PROGRAM PRG_LARS_ValidationAsConfirmation
VAR
	rtrigNewOuterArrived					: R_TRIG;
	bNewOuterIsProccesing				: BOOL;
	tonValidationTimout					: TON;
	bValidationTimeout					: BOOL;
	bValidationTimeoutReset				: BOOL;
	fbTimeoutCounter						: CTU;
	nCount									: WORD;
	fbPerformance							: FB_Interval;

	bOuterValidationCameraTrigger			: BOOL;
	aOuterValidationCamera				:  ARRAY[1..2] OF FB_SCANNER_CameraSelect;
	stOuterValidationCameraStatus		: ST_SCANNER;
	(*stOuterValidationCameraOptions		: ST_SCANNER_Options := (eScannerType := E_MV_420_FULL, nImageBuffer := 1, nExpectedResp := 2);*)
	aOuterValidationEvaluation			: ARRAY[1..2] OF FB_SCANNER_Evaluation;

	fbValidationCameraOut				: FB_OUTER_ValidationCameraOut;
	fbCheckForDuplicateOuterValidation	: FB_OUTER_CheckDuplicateStatus;

	(*rtrigOuterValidationCameraDone		: R_TRIG;
	bOuterValidationCameraDone			: BOOL;*)
	bDataReadyForValidation				: BOOL;
	bQAReject								: BOOL;

	sLastImageLableString				: T_OUTER_Barcode;

	fbMoveOuterData						: FB_OUTER_MoveOuterStatus;
	fbCompleteDataFromConfirmation	: FB_OUTER_CompleteDataFromDB_SingleCam;
	fbMETSValidateOuterForReject			: FB_OUTER_ValidateOuterForReject;
	tofValidateOuterDoneForHMI			: TOF;
	fbMasterListUpdate					: FB_OUTER_MasterListUpdate;

	stLastOuterCompleted					: ST_OUTER_Status;
	sLastReadOuterBarcode				: T_OUTER_Barcode;
	sLastReadConfPackCode1				: T_PACK_Barcode;
	nOutersCompleted						: UDINT;
	bDoneInfo								: BOOL;

	rtrigSetOuterValidationOK			: R_TRIG;
	rtrigSetOuterValidationNOK		: R_TRIG;

	rsOuterRejectStation 				: RS;
	rsOuterRejectConfirmation 		: RS;

	rtrigResetValidationStatus			: R_TRIG;

	sRejectCode						: STRING(255);
	fbArchiveInvalidOuters			: FB_OUTER_ArchiveInvalidOuters;
	aReasonForReject					: ARRAY[0..50] OF STRING(255);
	bClearList							: BOOL;

	fbOuterProduced					: FB_KPI_GenericEfficiency;
	fbOuterInspection					: FB_KPI_OutersEfficiency;

	fbOuterLevelCounter				: FB_KPI_OuterLevelCounter;

	fbQARejectCounter				: FB_CTU32;
	fbOuterValidationIndexOK			: FB_CTU32;

	ctuConsecutiveOuterRejects		: CTU;
	nActualCount						: WORD;

	stDummyImageData			: ST_SCANNER_ImageData;		(* image data structure *)
	aDistanceCheck				: ARRAY[1..2] OF FB_TimeDistance;
	bResetCTU						: BOOL;
END_VAR
VAR // added by the converter: edge detectors and wires of the graphical bodies
    _w1 : BOOL;
END_VAR

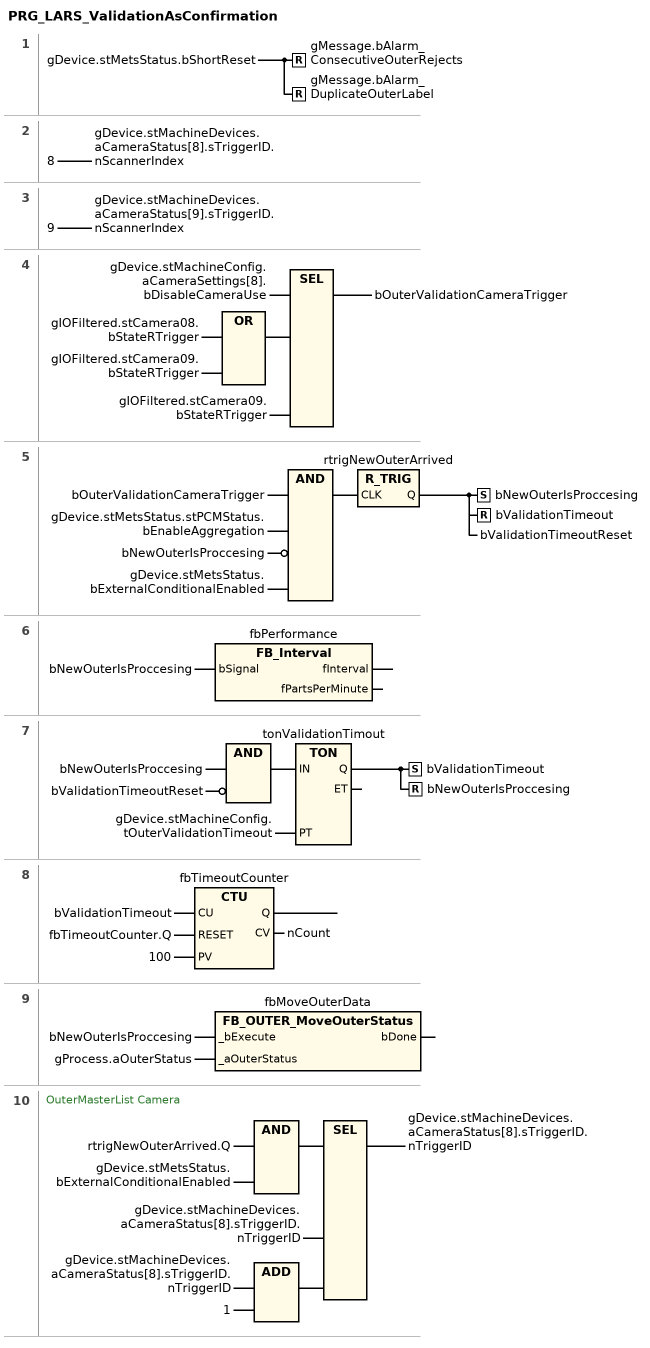
// NETWORK 1
gMessage.bAlarm_ConsecutiveOuterRejects R= gDevice.stMetsStatus.bShortReset;
gMessage.bAlarm_DuplicateOuterLabel R= gDevice.stMetsStatus.bShortReset;

// NETWORK 2
gDevice.stMachineDevices.aCameraStatus[8].sTriggerID.nScannerIndex := 8;

// NETWORK 3
gDevice.stMachineDevices.aCameraStatus[9].sTriggerID.nScannerIndex := 9;

// NETWORK 4
bOuterValidationCameraTrigger := SEL(gDevice.stMachineConfig.aCameraSettings[8].bDisableCameraUse, gIOFiltered.stCamera08.bStateRTrigger OR gIOFiltered.stCamera09.bStateRTrigger, gIOFiltered.stCamera09.bStateRTrigger);

// NETWORK 5
rtrigNewOuterArrived(CLK := bOuterValidationCameraTrigger AND gDevice.stMetsStatus.stPCMStatus.bEnableAggregation AND NOT bNewOuterIsProccesing AND gDevice.stMetsStatus.bExternalConditionalEnabled); // R_TRIG
bNewOuterIsProccesing S= rtrigNewOuterArrived.Q;
bValidationTimeout R= rtrigNewOuterArrived.Q;
bValidationTimeoutReset := rtrigNewOuterArrived.Q;

// NETWORK 6
fbPerformance(bSignal := bNewOuterIsProccesing); // FB_Interval

// NETWORK 7
tonValidationTimout(IN := bNewOuterIsProccesing AND NOT bValidationTimeoutReset, PT := gDevice.stMachineConfig.tOuterValidationTimeout); // TON
bValidationTimeout S= tonValidationTimout.Q;
bNewOuterIsProccesing R= tonValidationTimout.Q;

// NETWORK 8
fbTimeoutCounter(CU := bValidationTimeout, RESET := fbTimeoutCounter.Q, PV := 100, CV => nCount); // CTU

// NETWORK 9
fbMoveOuterData(_bExecute := bNewOuterIsProccesing, _aOuterStatus := gProcess.aOuterStatus); // FB_OUTER_MoveOuterStatus

// NETWORK 10
// OuterMasterList Camera
gDevice.stMachineDevices.aCameraStatus[8].sTriggerID.nTriggerID := SEL(rtrigNewOuterArrived.Q AND gDevice.stMetsStatus.bExternalConditionalEnabled, gDevice.stMachineDevices.aCameraStatus[8].sTriggerID.nTriggerID, gDevice.stMachineDevices.aCameraStatus[8].sTriggerID.nTriggerID + 1);

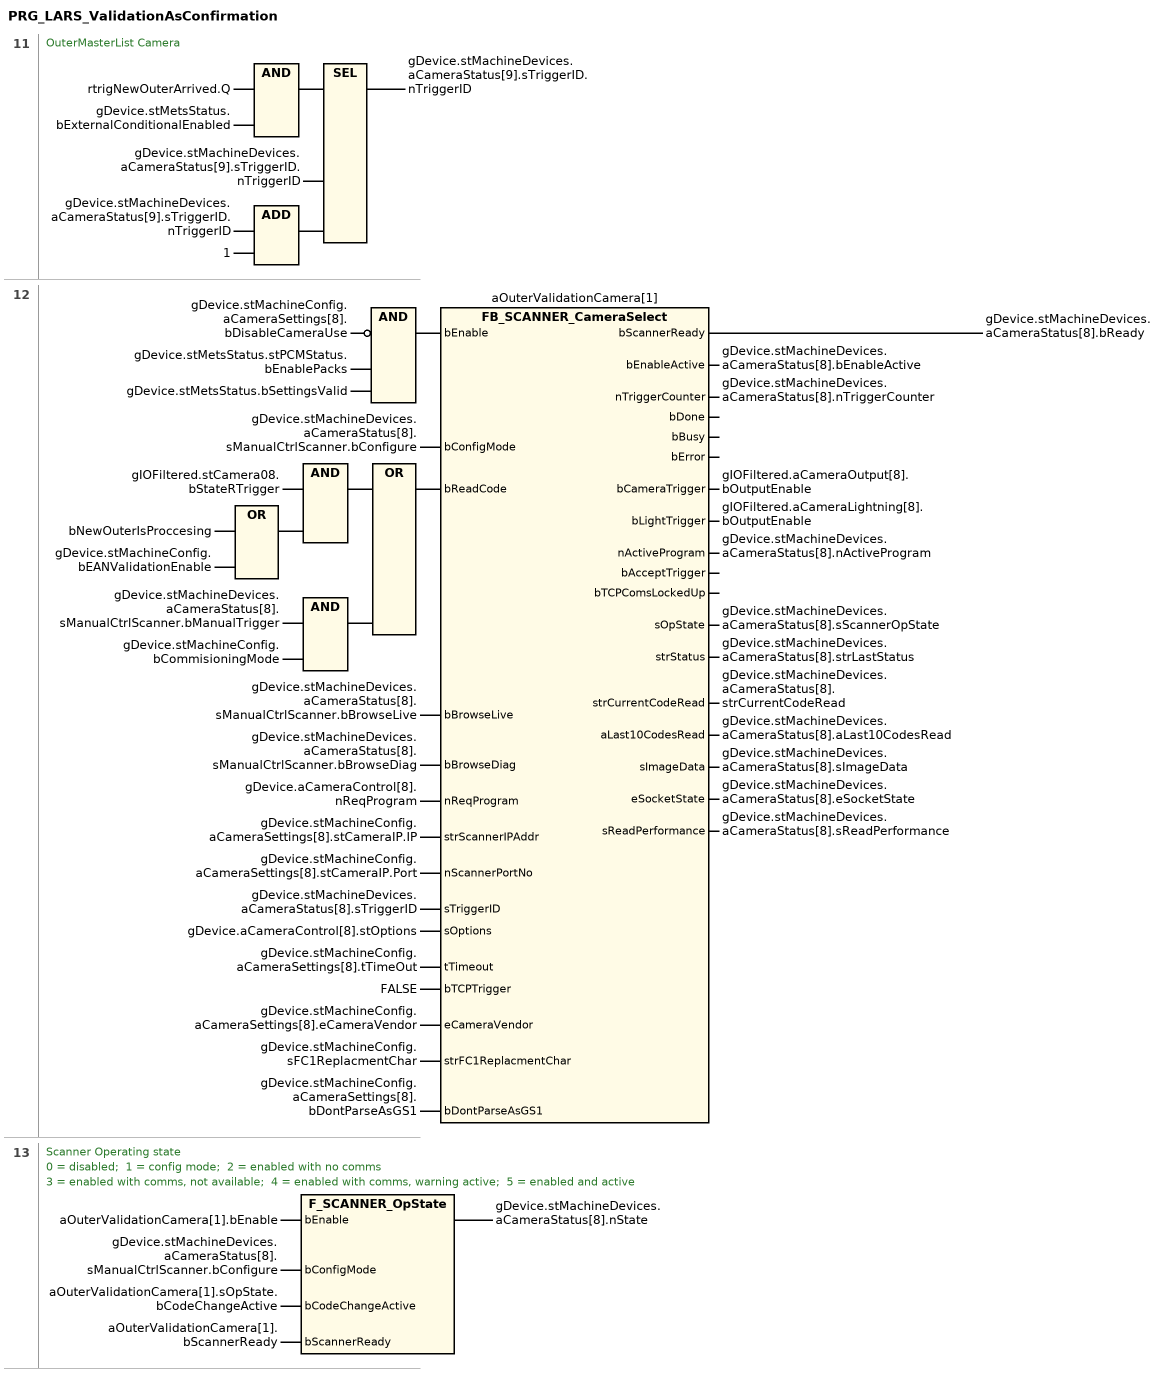
// NETWORK 11
// OuterMasterList Camera
gDevice.stMachineDevices.aCameraStatus[9].sTriggerID.nTriggerID := SEL(rtrigNewOuterArrived.Q AND gDevice.stMetsStatus.bExternalConditionalEnabled, gDevice.stMachineDevices.aCameraStatus[9].sTriggerID.nTriggerID, gDevice.stMachineDevices.aCameraStatus[9].sTriggerID.nTriggerID + 1);

// NETWORK 12
aOuterValidationCamera[1](
    bEnable := NOT gDevice.stMachineConfig.aCameraSettings[8].bDisableCameraUse AND gDevice.stMetsStatus.stPCMStatus.bEnablePacks AND gDevice.stMetsStatus.bSettingsValid,
    bConfigMode := gDevice.stMachineDevices.aCameraStatus[8].sManualCtrlScanner.bConfigure,
    bReadCode := gIOFiltered.stCamera08.bStateRTrigger AND (bNewOuterIsProccesing OR gDevice.stMachineConfig.bEANValidationEnable) OR gDevice.stMachineDevices.aCameraStatus[8].sManualCtrlScanner.bManualTrigger AND gDevice.stMachineConfig.bCommisioningMode,
    bBrowseLive := gDevice.stMachineDevices.aCameraStatus[8].sManualCtrlScanner.bBrowseLive,
    bBrowseDiag := gDevice.stMachineDevices.aCameraStatus[8].sManualCtrlScanner.bBrowseDiag,
    nReqProgram := gDevice.aCameraControl[8].nReqProgram,
    strScannerIPAddr := gDevice.stMachineConfig.aCameraSettings[8].stCameraIP.IP,
    nScannerPortNo := gDevice.stMachineConfig.aCameraSettings[8].stCameraIP.Port,
    sTriggerID := gDevice.stMachineDevices.aCameraStatus[8].sTriggerID,
    sOptions := gDevice.aCameraControl[8].stOptions,
    tTimeout := gDevice.stMachineConfig.aCameraSettings[8].tTimeOut,
    bTCPTrigger := FALSE,
    eCameraVendor := gDevice.stMachineConfig.aCameraSettings[8].eCameraVendor,
    strFC1ReplacmentChar := gDevice.stMachineConfig.sFC1ReplacmentChar,
    bDontParseAsGS1 := gDevice.stMachineConfig.aCameraSettings[8].bDontParseAsGS1,
    bEnableActive => gDevice.stMachineDevices.aCameraStatus[8].bEnableActive,
    nTriggerCounter => gDevice.stMachineDevices.aCameraStatus[8].nTriggerCounter,
    bCameraTrigger => gIOFiltered.aCameraOutput[8].bOutputEnable,
    bLightTrigger => gIOFiltered.aCameraLightning[8].bOutputEnable,
    nActiveProgram => gDevice.stMachineDevices.aCameraStatus[8].nActiveProgram,
    sOpState => gDevice.stMachineDevices.aCameraStatus[8].sScannerOpState,
    strStatus => gDevice.stMachineDevices.aCameraStatus[8].strLastStatus,
    strCurrentCodeRead => gDevice.stMachineDevices.aCameraStatus[8].strCurrentCodeRead,
    aLast10CodesRead => gDevice.stMachineDevices.aCameraStatus[8].aLast10CodesRead,
    sImageData => gDevice.stMachineDevices.aCameraStatus[8].sImageData,
    eSocketState => gDevice.stMachineDevices.aCameraStatus[8].eSocketState,
    sReadPerformance => gDevice.stMachineDevices.aCameraStatus[8].sReadPerformance); // FB_SCANNER_CameraSelect
gDevice.stMachineDevices.aCameraStatus[8].bReady := aOuterValidationCamera[1].bScannerReady;

// NETWORK 13
// 					Scanner Operating state
// 0 = disabled;  1 = config mode;  2 = enabled with no comms
// 3 = enabled with comms, not available;  4 = enabled with comms, warning active;  5 = enabled and active
//
gDevice.stMachineDevices.aCameraStatus[8].nState := F_SCANNER_OpState(bEnable := aOuterValidationCamera[1].bEnable, bConfigMode := gDevice.stMachineDevices.aCameraStatus[8].sManualCtrlScanner.bConfigure, bCodeChangeActive := aOuterValidationCamera[1].sOpState.bCodeChangeActive, bScannerReady := aOuterValidationCamera[1].bScannerReady);

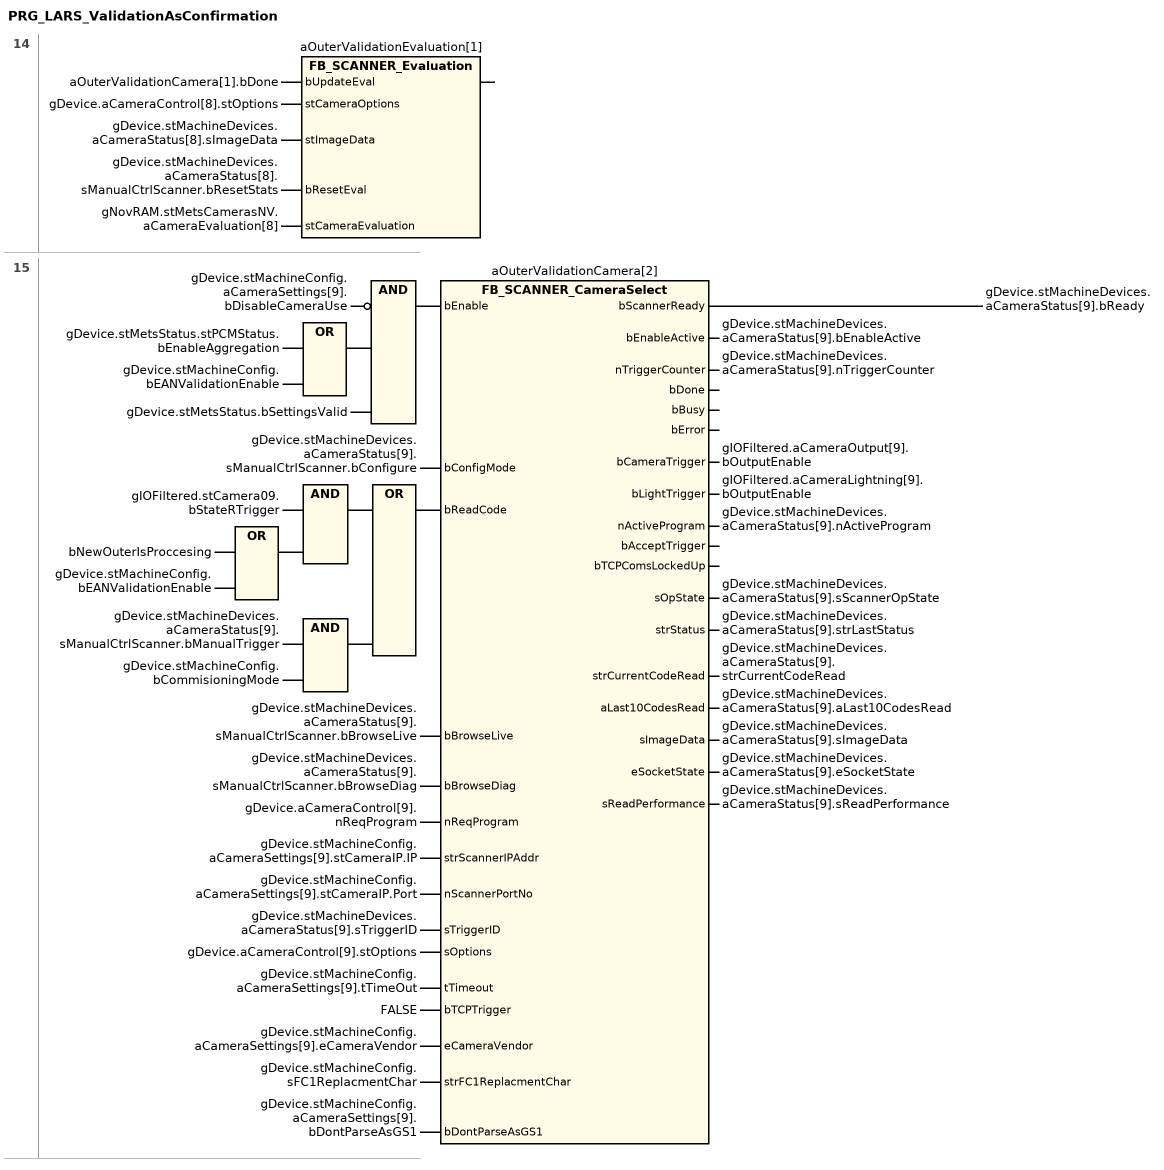
// NETWORK 14
aOuterValidationEvaluation[1](
    bUpdateEval := aOuterValidationCamera[1].bDone,
    stCameraOptions := gDevice.aCameraControl[8].stOptions,
    stImageData := gDevice.stMachineDevices.aCameraStatus[8].sImageData,
    bResetEval := gDevice.stMachineDevices.aCameraStatus[8].sManualCtrlScanner.bResetStats,
    stCameraEvaluation := gNovRAM.stMetsCamerasNV.aCameraEvaluation[8]); // FB_SCANNER_Evaluation

// NETWORK 15
aOuterValidationCamera[2](
    bEnable := NOT gDevice.stMachineConfig.aCameraSettings[9].bDisableCameraUse AND (gDevice.stMetsStatus.stPCMStatus.bEnableAggregation OR gDevice.stMachineConfig.bEANValidationEnable) AND gDevice.stMetsStatus.bSettingsValid,
    bConfigMode := gDevice.stMachineDevices.aCameraStatus[9].sManualCtrlScanner.bConfigure,
    bReadCode := gIOFiltered.stCamera09.bStateRTrigger AND (bNewOuterIsProccesing OR gDevice.stMachineConfig.bEANValidationEnable) OR gDevice.stMachineDevices.aCameraStatus[9].sManualCtrlScanner.bManualTrigger AND gDevice.stMachineConfig.bCommisioningMode,
    bBrowseLive := gDevice.stMachineDevices.aCameraStatus[9].sManualCtrlScanner.bBrowseLive,
    bBrowseDiag := gDevice.stMachineDevices.aCameraStatus[9].sManualCtrlScanner.bBrowseDiag,
    nReqProgram := gDevice.aCameraControl[9].nReqProgram,
    strScannerIPAddr := gDevice.stMachineConfig.aCameraSettings[9].stCameraIP.IP,
    nScannerPortNo := gDevice.stMachineConfig.aCameraSettings[9].stCameraIP.Port,
    sTriggerID := gDevice.stMachineDevices.aCameraStatus[9].sTriggerID,
    sOptions := gDevice.aCameraControl[9].stOptions,
    tTimeout := gDevice.stMachineConfig.aCameraSettings[9].tTimeOut,
    bTCPTrigger := FALSE,
    eCameraVendor := gDevice.stMachineConfig.aCameraSettings[9].eCameraVendor,
    strFC1ReplacmentChar := gDevice.stMachineConfig.sFC1ReplacmentChar,
    bDontParseAsGS1 := gDevice.stMachineConfig.aCameraSettings[9].bDontParseAsGS1,
    bEnableActive => gDevice.stMachineDevices.aCameraStatus[9].bEnableActive,
    nTriggerCounter => gDevice.stMachineDevices.aCameraStatus[9].nTriggerCounter,
    bCameraTrigger => gIOFiltered.aCameraOutput[9].bOutputEnable,
    bLightTrigger => gIOFiltered.aCameraLightning[9].bOutputEnable,
    nActiveProgram => gDevice.stMachineDevices.aCameraStatus[9].nActiveProgram,
    sOpState => gDevice.stMachineDevices.aCameraStatus[9].sScannerOpState,
    strStatus => gDevice.stMachineDevices.aCameraStatus[9].strLastStatus,
    strCurrentCodeRead => gDevice.stMachineDevices.aCameraStatus[9].strCurrentCodeRead,
    aLast10CodesRead => gDevice.stMachineDevices.aCameraStatus[9].aLast10CodesRead,
    sImageData => gDevice.stMachineDevices.aCameraStatus[9].sImageData,
    eSocketState => gDevice.stMachineDevices.aCameraStatus[9].eSocketState,
    sReadPerformance => gDevice.stMachineDevices.aCameraStatus[9].sReadPerformance); // FB_SCANNER_CameraSelect
gDevice.stMachineDevices.aCameraStatus[9].bReady := aOuterValidationCamera[2].bScannerReady;

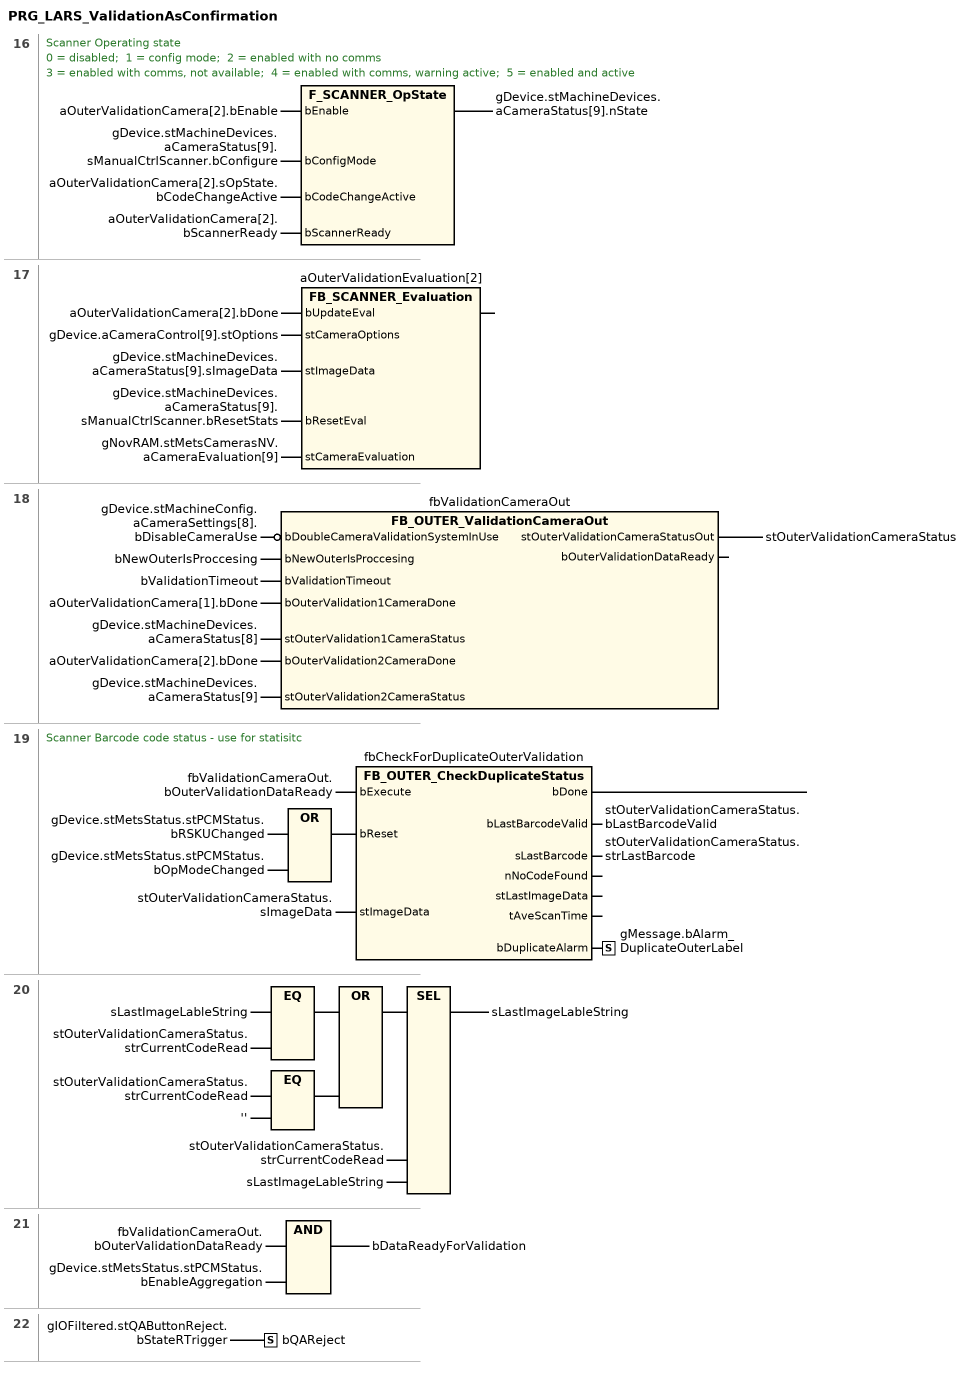
// NETWORK 16
// 					Scanner Operating state
// 0 = disabled;  1 = config mode;  2 = enabled with no comms
// 3 = enabled with comms, not available;  4 = enabled with comms, warning active;  5 = enabled and active
//
gDevice.stMachineDevices.aCameraStatus[9].nState := F_SCANNER_OpState(bEnable := aOuterValidationCamera[2].bEnable, bConfigMode := gDevice.stMachineDevices.aCameraStatus[9].sManualCtrlScanner.bConfigure, bCodeChangeActive := aOuterValidationCamera[2].sOpState.bCodeChangeActive, bScannerReady := aOuterValidationCamera[2].bScannerReady);

// NETWORK 17
aOuterValidationEvaluation[2](
    bUpdateEval := aOuterValidationCamera[2].bDone,
    stCameraOptions := gDevice.aCameraControl[9].stOptions,
    stImageData := gDevice.stMachineDevices.aCameraStatus[9].sImageData,
    bResetEval := gDevice.stMachineDevices.aCameraStatus[9].sManualCtrlScanner.bResetStats,
    stCameraEvaluation := gNovRAM.stMetsCamerasNV.aCameraEvaluation[9]); // FB_SCANNER_Evaluation

// NETWORK 18
fbValidationCameraOut(
    bDoubleCameraValidationSystemInUse := NOT gDevice.stMachineConfig.aCameraSettings[8].bDisableCameraUse,
    bNewOuterIsProccesing := bNewOuterIsProccesing,
    bValidationTimeout := bValidationTimeout,
    bOuterValidation1CameraDone := aOuterValidationCamera[1].bDone,
    stOuterValidation1CameraStatus := gDevice.stMachineDevices.aCameraStatus[8],
    bOuterValidation2CameraDone := aOuterValidationCamera[2].bDone,
    stOuterValidation2CameraStatus := gDevice.stMachineDevices.aCameraStatus[9]); // FB_OUTER_ValidationCameraOut
stOuterValidationCameraStatus := fbValidationCameraOut.stOuterValidationCameraStatusOut;

// NETWORK 19
// Scanner Barcode code status - use for statisitc
fbCheckForDuplicateOuterValidation(
    bExecute := fbValidationCameraOut.bOuterValidationDataReady,
    bReset := gDevice.stMetsStatus.stPCMStatus.bRSKUChanged OR gDevice.stMetsStatus.stPCMStatus.bOpModeChanged,
    stImageData := stOuterValidationCameraStatus.sImageData,
    bLastBarcodeValid => stOuterValidationCameraStatus.bLastBarcodeValid,
    sLastBarcode => stOuterValidationCameraStatus.strLastBarcode); // FB_OUTER_CheckDuplicateStatus
gMessage.bAlarm_DuplicateOuterLabel S= fbCheckForDuplicateOuterValidation.bDuplicateAlarm;

// NETWORK 20
sLastImageLableString := SEL(sLastImageLableString = stOuterValidationCameraStatus.strCurrentCodeRead OR stOuterValidationCameraStatus.strCurrentCodeRead = '', stOuterValidationCameraStatus.strCurrentCodeRead, sLastImageLableString);

// NETWORK 21
bDataReadyForValidation := fbValidationCameraOut.bOuterValidationDataReady AND gDevice.stMetsStatus.stPCMStatus.bEnableAggregation;

// NETWORK 22
bQAReject S= gIOFiltered.stQAButtonReject.bStateRTrigger;

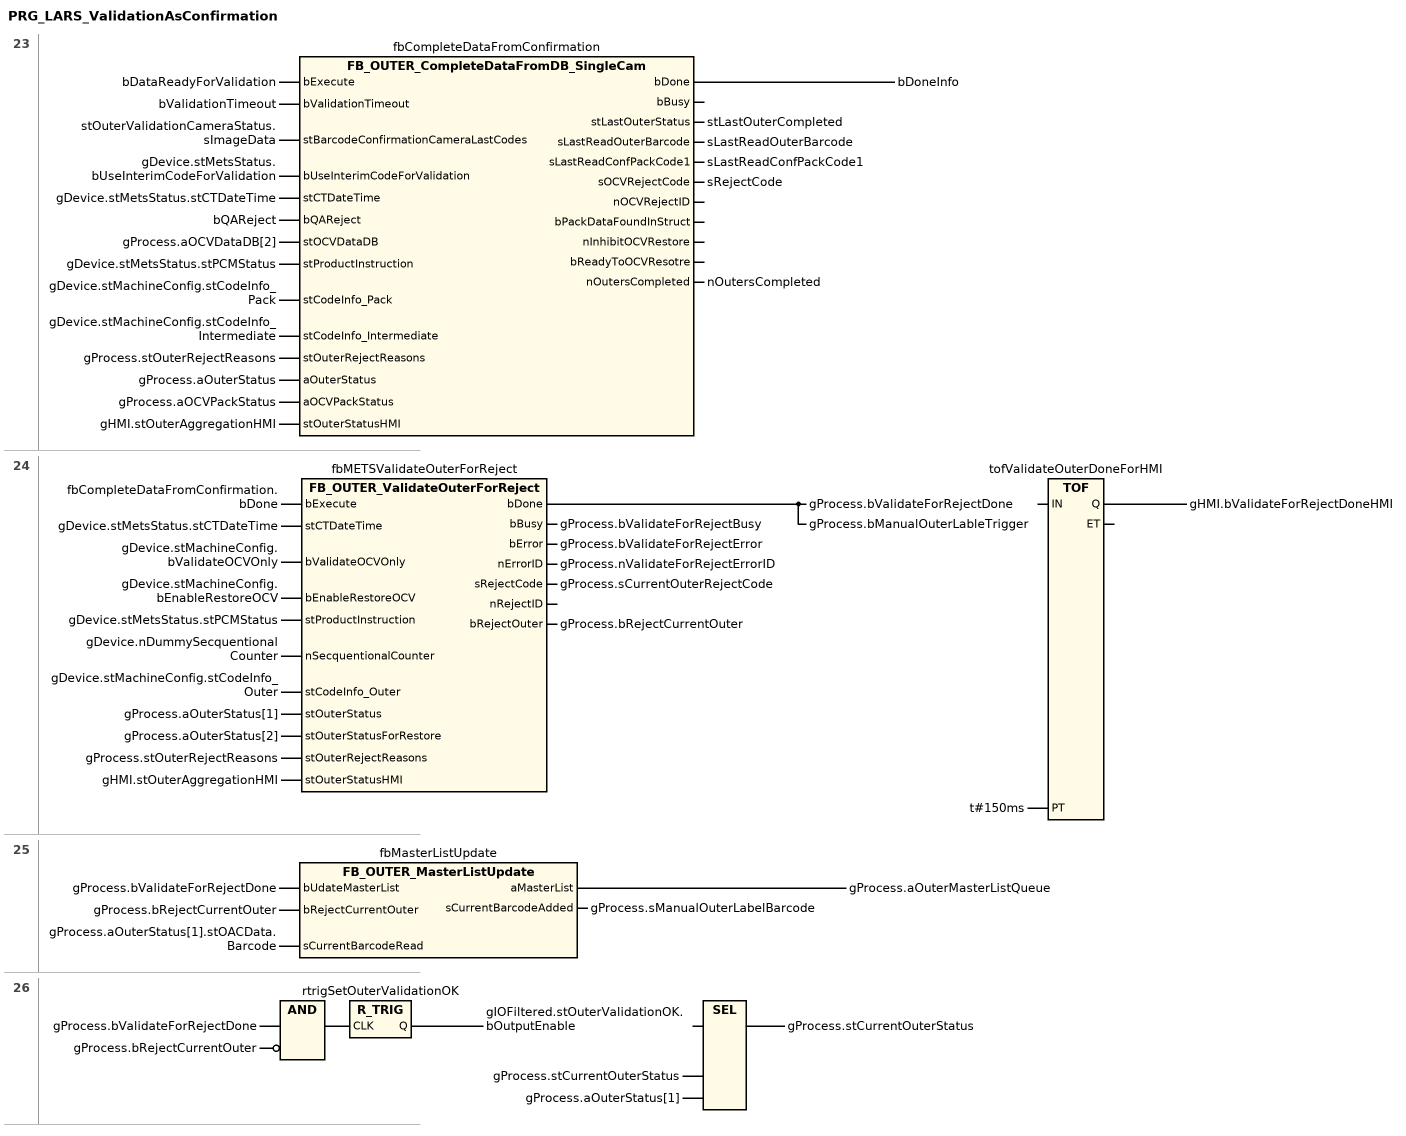
// NETWORK 23
fbCompleteDataFromConfirmation(
    bExecute := bDataReadyForValidation,
    bValidationTimeout := bValidationTimeout,
    stBarcodeConfirmationCameraLastCodes := stOuterValidationCameraStatus.sImageData,
    bUseInterimCodeForValidation := gDevice.stMetsStatus.bUseInterimCodeForValidation,
    stCTDateTime := gDevice.stMetsStatus.stCTDateTime,
    bQAReject := bQAReject,
    stOCVDataDB := gProcess.aOCVDataDB[2],
    stProductInstruction := gDevice.stMetsStatus.stPCMStatus,
    stCodeInfo_Pack := gDevice.stMachineConfig.stCodeInfo_Pack,
    stCodeInfo_Intermediate := gDevice.stMachineConfig.stCodeInfo_Intermediate,
    stOuterRejectReasons := gProcess.stOuterRejectReasons,
    aOuterStatus := gProcess.aOuterStatus,
    aOCVPackStatus := gProcess.aOCVPackStatus,
    stOuterStatusHMI := gHMI.stOuterAggregationHMI,
    stLastOuterStatus => stLastOuterCompleted,
    sLastReadOuterBarcode => sLastReadOuterBarcode,
    sLastReadConfPackCode1 => sLastReadConfPackCode1,
    sOCVRejectCode => sRejectCode,
    nOutersCompleted => nOutersCompleted); // FB_OUTER_CompleteDataFromDB_SingleCam
bDoneInfo := fbCompleteDataFromConfirmation.bDone;

// NETWORK 24
fbMETSValidateOuterForReject(
    bExecute := fbCompleteDataFromConfirmation.bDone,
    stCTDateTime := gDevice.stMetsStatus.stCTDateTime,
    bValidateOCVOnly := gDevice.stMachineConfig.bValidateOCVOnly,
    bEnableRestoreOCV := gDevice.stMachineConfig.bEnableRestoreOCV,
    stProductInstruction := gDevice.stMetsStatus.stPCMStatus,
    nSecquentionalCounter := gDevice.nDummySecquentionalCounter,
    stCodeInfo_Outer := gDevice.stMachineConfig.stCodeInfo_Outer,
    stOuterStatus := gProcess.aOuterStatus[1],
    stOuterStatusForRestore := gProcess.aOuterStatus[2],
    stOuterRejectReasons := gProcess.stOuterRejectReasons,
    stOuterStatusHMI := gHMI.stOuterAggregationHMI,
    bBusy => gProcess.bValidateForRejectBusy,
    bError => gProcess.bValidateForRejectError,
    nErrorID => gProcess.nValidateForRejectErrorID,
    sRejectCode => gProcess.sCurrentOuterRejectCode,
    bRejectOuter => gProcess.bRejectCurrentOuter); // FB_OUTER_ValidateOuterForReject
gProcess.bValidateForRejectDone := fbMETSValidateOuterForReject.bDone;
gProcess.bManualOuterLableTrigger := fbMETSValidateOuterForReject.bDone;
tofValidateOuterDoneForHMI(IN := fbMETSValidateOuterForReject.bDone, PT := t#150ms); // TOF
gHMI.bValidateForRejectDoneHMI := tofValidateOuterDoneForHMI.Q;

// NETWORK 25
fbMasterListUpdate(
    bUdateMasterList := gProcess.bValidateForRejectDone,
    bRejectCurrentOuter := gProcess.bRejectCurrentOuter,
    sCurrentBarcodeRead := gProcess.aOuterStatus[1].stOACData.Barcode,
    sCurrentBarcodeAdded => gProcess.sManualOuterLabelBarcode); // FB_OUTER_MasterListUpdate
gProcess.aOuterMasterListQueue := fbMasterListUpdate.aMasterList;

// NETWORK 26
rtrigSetOuterValidationOK(CLK := gProcess.bValidateForRejectDone AND NOT gProcess.bRejectCurrentOuter); // R_TRIG
gIOFiltered.stOuterValidationOK.bOutputEnable := rtrigSetOuterValidationOK.Q;
gProcess.stCurrentOuterStatus := SEL(rtrigSetOuterValidationOK.Q, gProcess.stCurrentOuterStatus, gProcess.aOuterStatus[1]);

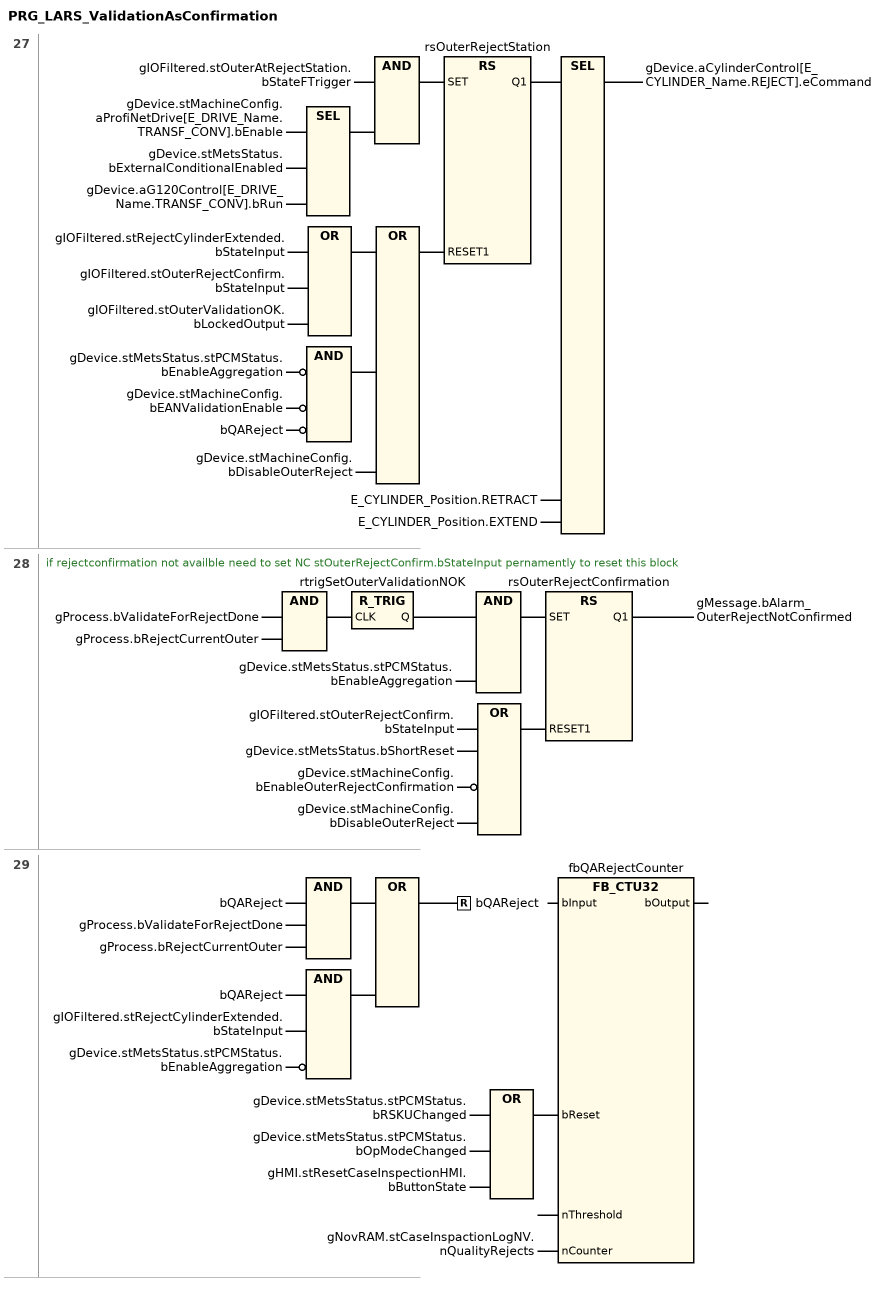
// NETWORK 27
rsOuterRejectStation(SET := gIOFiltered.stOuterAtRejectStation.bStateFTrigger AND SEL(gDevice.stMachineConfig.aProfiNetDrive[E_DRIVE_Name.TRANSF_CONV].bEnable, gDevice.stMetsStatus.bExternalConditionalEnabled, gDevice.aG120Control[E_DRIVE_Name.TRANSF_CONV].bRun), RESET1 := (gIOFiltered.stRejectCylinderExtended.bStateInput OR gIOFiltered.stOuterRejectConfirm.bStateInput OR gIOFiltered.stOuterValidationOK.bLockedOutput) OR NOT gDevice.stMetsStatus.stPCMStatus.bEnableAggregation AND NOT gDevice.stMachineConfig.bEANValidationEnable AND NOT bQAReject OR gDevice.stMachineConfig.bDisableOuterReject); // RS
gDevice.aCylinderControl[E_CYLINDER_Name.REJECT].eCommand := SEL(rsOuterRejectStation.Q1, E_CYLINDER_Position.RETRACT, E_CYLINDER_Position.EXTEND);

// NETWORK 28
// if rejectconfirmation not availble need to set NC stOuterRejectConfirm.bStateInput pernamently to reset this block
rtrigSetOuterValidationNOK(CLK := gProcess.bValidateForRejectDone AND gProcess.bRejectCurrentOuter); // R_TRIG
rsOuterRejectConfirmation(SET := rtrigSetOuterValidationNOK.Q AND gDevice.stMetsStatus.stPCMStatus.bEnableAggregation, RESET1 := gIOFiltered.stOuterRejectConfirm.bStateInput OR gDevice.stMetsStatus.bShortReset OR NOT gDevice.stMachineConfig.bEnableOuterRejectConfirmation OR gDevice.stMachineConfig.bDisableOuterReject); // RS
gMessage.bAlarm_OuterRejectNotConfirmed := rsOuterRejectConfirmation.Q1;

// NETWORK 29
_w1 := bQAReject AND gProcess.bValidateForRejectDone AND gProcess.bRejectCurrentOuter OR bQAReject AND gIOFiltered.stRejectCylinderExtended.bStateInput AND NOT gDevice.stMetsStatus.stPCMStatus.bEnableAggregation;
bQAReject R= _w1;
fbQARejectCounter(
    bInput := _w1,
    bReset := gDevice.stMetsStatus.stPCMStatus.bRSKUChanged OR gDevice.stMetsStatus.stPCMStatus.bOpModeChanged OR gHMI.stResetCaseInspectionHMI.bButtonState,
    nCounter := gNovRAM.stCaseInspactionLogNV.nQualityRejects); // FB_CTU32

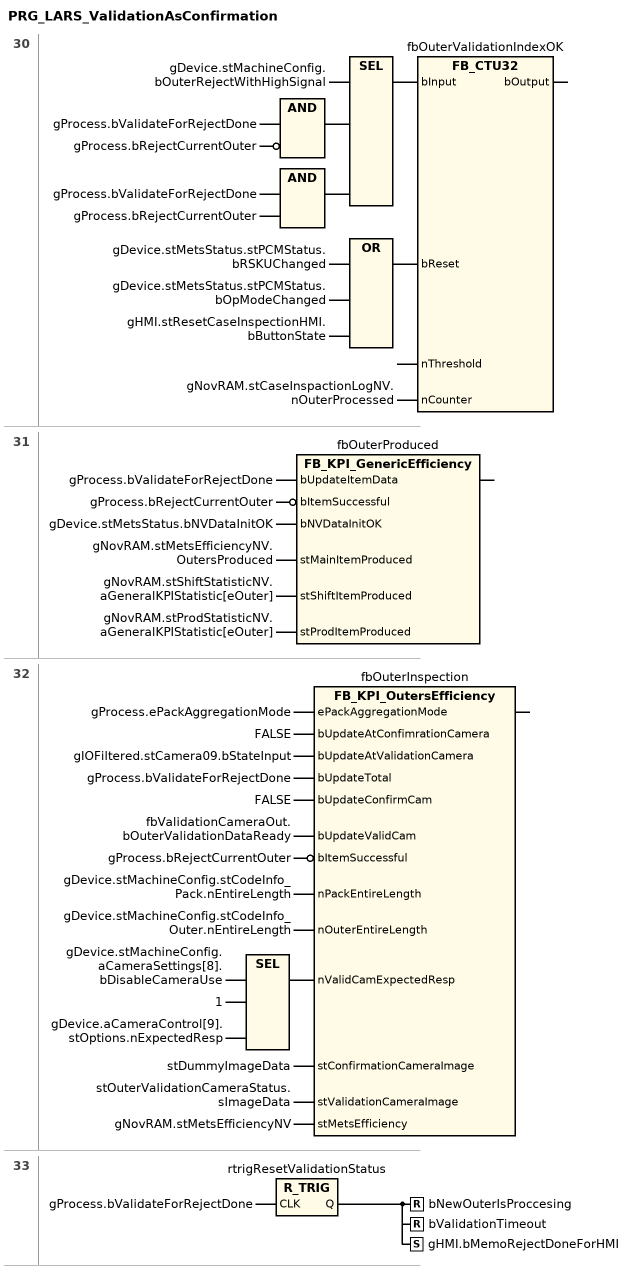
// NETWORK 30
fbOuterValidationIndexOK(
    bInput := SEL(gDevice.stMachineConfig.bOuterRejectWithHighSignal, gProcess.bValidateForRejectDone AND NOT gProcess.bRejectCurrentOuter, gProcess.bValidateForRejectDone AND gProcess.bRejectCurrentOuter),
    bReset := gDevice.stMetsStatus.stPCMStatus.bRSKUChanged OR gDevice.stMetsStatus.stPCMStatus.bOpModeChanged OR gHMI.stResetCaseInspectionHMI.bButtonState,
    nCounter := gNovRAM.stCaseInspactionLogNV.nOuterProcessed); // FB_CTU32

// NETWORK 31
fbOuterProduced(
    bUpdateItemData := gProcess.bValidateForRejectDone,
    bItemSuccessful := NOT gProcess.bRejectCurrentOuter,
    bNVDataInitOK := gDevice.stMetsStatus.bNVDataInitOK,
    stMainItemProduced := gNovRAM.stMetsEfficiencyNV.OutersProduced,
    stShiftItemProduced := gNovRAM.stShiftStatisticNV.aGeneralKPIStatistic[eOuter],
    stProdItemProduced := gNovRAM.stProdStatisticNV.aGeneralKPIStatistic[eOuter]); // FB_KPI_GenericEfficiency

// NETWORK 32
fbOuterInspection(
    ePackAggregationMode := gProcess.ePackAggregationMode,
    bUpdateAtConfimrationCamera := FALSE,
    bUpdateAtValidationCamera := gIOFiltered.stCamera09.bStateInput,
    bUpdateTotal := gProcess.bValidateForRejectDone,
    bUpdateConfirmCam := FALSE,
    bUpdateValidCam := fbValidationCameraOut.bOuterValidationDataReady,
    bItemSuccessful := NOT gProcess.bRejectCurrentOuter,
    nPackEntireLength := gDevice.stMachineConfig.stCodeInfo_Pack.nEntireLength,
    nOuterEntireLength := gDevice.stMachineConfig.stCodeInfo_Outer.nEntireLength,
    nValidCamExpectedResp := SEL(gDevice.stMachineConfig.aCameraSettings[8].bDisableCameraUse, 1, gDevice.aCameraControl[9].stOptions.nExpectedResp),
    stConfirmationCameraImage := stDummyImageData,
    stValidationCameraImage := stOuterValidationCameraStatus.sImageData,
    stMetsEfficiency := gNovRAM.stMetsEfficiencyNV); // FB_KPI_OutersEfficiency

// NETWORK 33
rtrigResetValidationStatus(CLK := gProcess.bValidateForRejectDone); // R_TRIG
bNewOuterIsProccesing R= rtrigResetValidationStatus.Q;
bValidationTimeout R= rtrigResetValidationStatus.Q;
gHMI.bMemoRejectDoneForHMI S= rtrigResetValidationStatus.Q;

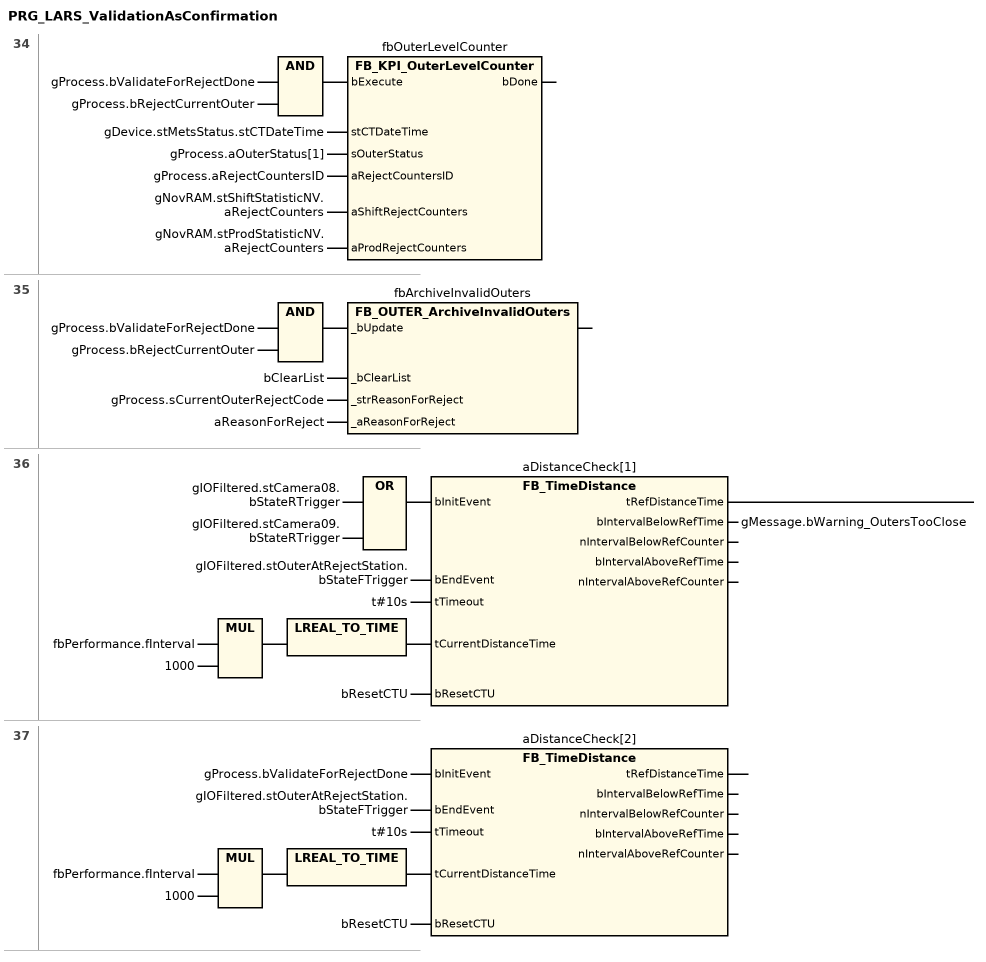
// NETWORK 34
fbOuterLevelCounter(
    bExecute := gProcess.bValidateForRejectDone AND gProcess.bRejectCurrentOuter,
    stCTDateTime := gDevice.stMetsStatus.stCTDateTime,
    sOuterStatus := gProcess.aOuterStatus[1],
    aRejectCountersID := gProcess.aRejectCountersID,
    aShiftRejectCounters := gNovRAM.stShiftStatisticNV.aRejectCounters,
    aProdRejectCounters := gNovRAM.stProdStatisticNV.aRejectCounters); // FB_KPI_OuterLevelCounter

// NETWORK 35
fbArchiveInvalidOuters(
    _bUpdate := gProcess.bValidateForRejectDone AND gProcess.bRejectCurrentOuter,
    _bClearList := bClearList,
    _strReasonForReject := gProcess.sCurrentOuterRejectCode,
    _aReasonForReject := aReasonForReject); // FB_OUTER_ArchiveInvalidOuters

// NETWORK 36
aDistanceCheck[1](
    bInitEvent := gIOFiltered.stCamera08.bStateRTrigger OR gIOFiltered.stCamera09.bStateRTrigger,
    bEndEvent := gIOFiltered.stOuterAtRejectStation.bStateFTrigger,
    tTimeout := t#10s,
    tCurrentDistanceTime := LREAL_TO_TIME(fbPerformance.fInterval * 1000),
    bResetCTU := bResetCTU,
    bIntervalBelowRefTime => gMessage.bWarning_OutersTooClose); // FB_TimeDistance

// NETWORK 37
aDistanceCheck[2](
    bInitEvent := gProcess.bValidateForRejectDone,
    bEndEvent := gIOFiltered.stOuterAtRejectStation.bStateFTrigger,
    tTimeout := t#10s,
    tCurrentDistanceTime := LREAL_TO_TIME(fbPerformance.fInterval * 1000),
    bResetCTU := bResetCTU); // FB_TimeDistance

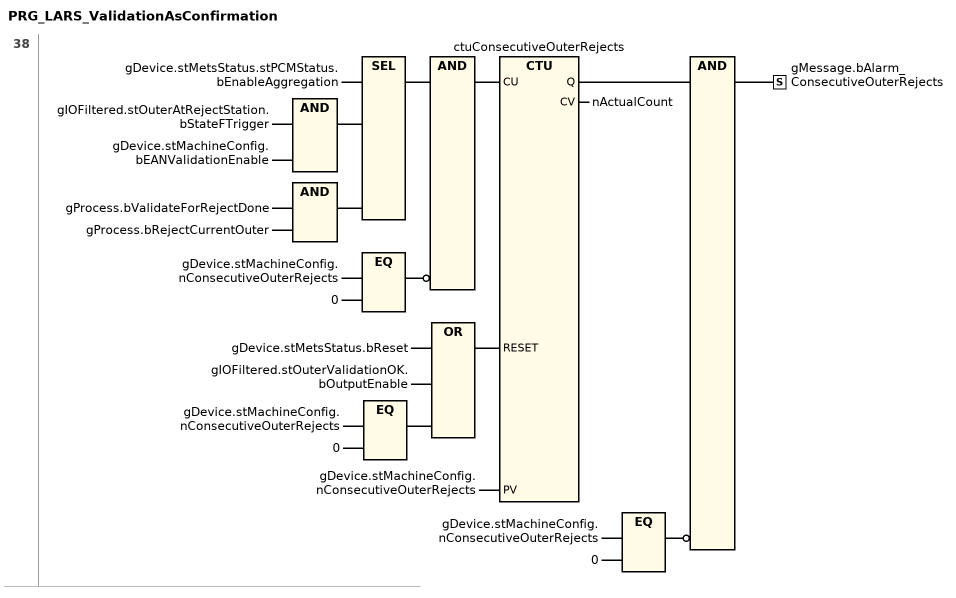
// NETWORK 38
ctuConsecutiveOuterRejects(
    CU := SEL(gDevice.stMetsStatus.stPCMStatus.bEnableAggregation, gIOFiltered.stOuterAtRejectStation.bStateFTrigger AND gDevice.stMachineConfig.bEANValidationEnable, gProcess.bValidateForRejectDone AND gProcess.bRejectCurrentOuter) AND NOT (gDevice.stMachineConfig.nConsecutiveOuterRejects = 0),
    RESET := gDevice.stMetsStatus.bReset OR gIOFiltered.stOuterValidationOK.bOutputEnable OR gDevice.stMachineConfig.nConsecutiveOuterRejects = 0,
    PV := gDevice.stMachineConfig.nConsecutiveOuterRejects,
    CV => nActualCount); // CTU
gMessage.bAlarm_ConsecutiveOuterRejects S= ctuConsecutiveOuterRejects.Q AND NOT (gDevice.stMachineConfig.nConsecutiveOuterRejects = 0);

END_PROGRAM

(* stored: Version 1.1.0.1
   POU PRG_LARS_ValidationAsConfirmation: Id {5ab1f032-982c-4d7e-a9da-173f6d64224b}, SpecialFunc None *)
